{attribute 'GeneratedUsingTerminal: EK1100-0000-0018'}
{attribute addProperty BoxType "EK1100-0000-0018"}
{attribute addProperty Id "Beckhoff_EKx9xxEK1122Beckhoff_EKx9xxEK1122_E046703E1090"}
{attribute addProperty CRC "2246922605"}
{attribute addProperty Size "1090"}
TYPE Beckhoff_EKx9xx_85ED516D EXTENDS EK1100_1FC0878B :
STRUCT
	{attribute addProperty Name "Beckhoff_EKx9xxEK1122"}
	{attribute addProperty PreviousPort "Beckhoff EKx9xx : B"}
	Beckhoff_EKx9xxEK1122 : Beckhoff_EKx9xxEK1122_E046703E;
END_STRUCT
END_TYPE

(* stored: Version 1.2.0.0, ProductVersion 3.1.4024.9
   DUT Beckhoff_EKx9xx_85ED516D: Id {ac14d686-8cb6-4d00-81e1-d77f5115ede0} *)
